FUNCTION_BLOCK FB_EventSubscriber2 IMPLEMENTS I_Observer
VAR_INPUT
	eventPublisher					: I_EventPublisher;
END_VAR
VAR
	_verbose						: BOOL := TRUE;
	_event							: INT;
	// Register after online change 
	registeredAtPublisher			: BOOL;

	breinit 						: BOOL; // reinit test marker
END_VAR

// Is there a valid publisher attached? 
IF eventPublisher=0	THEN
	RETURN;
END_IF

// Did we already register in the publisher?
IF NOT registeredAtPublisher	THEN
	registeredAtPublisher := eventPublisher.attach(THIS^);
END_IF

{attribute 'call_after_online_change_slot' := '0'}
METHOD PRIVATE fbreinit

(*	!!!!!!!!!!!!!!!!!!!!!!!!!!!!!!!!!
   	THIS METHOD is force called after every online change 
   	!= the fb_reinit system call that will be called after the instance of the concerned function block has been copied 
 	(during an online change after modifications in the function block declaration)

	This is necessary since both observer en observee 
	!!!!!!!!!!!!!!!!!!!!!!!!!!!!!!!!!	*)
registeredAtPublisher := FALSE;
breinit:=not breinit; // flip the test marker
END_METHOD

METHOD PRIVATE message : BOOL
VAR_INPUT
	dintArg						: DINT;
END_VAR
// Log message
IF _verbose  THEN
	ADSLOGDINT(
		msgCtrlMask := ADSLOG_MSGTYPE_HINT OR ADSLOG_MSGTYPE_LOG, // ADSLOG_MSGTYPE_ERROR OR ADSLOG_MSGTYPE_LOG, 
		msgFmtStr 	:= 'Subscriber 2 knows the value changed to %d',
		dintArg 	:= dintArg
		);
END_IF
END_METHOD

METHOD update : BOOL
// the publisher mentions an update, fetch the data
_event := eventPublisher.event;
message(TO_DINT(_event));
END_METHOD

END_FUNCTION_BLOCK

(* stored: Version 1.1.0.1, ProductVersion 3.1.4024.11
   POU FB_EventSubscriber2: Id {78948430-835f-4189-b81a-4f54b3428e0d}, SpecialFunc None
   Method fbreinit: Id {4f4019a2-6dab-4552-accd-abde4ac41c58}
   Method message: Id {89c2fe32-3b54-4706-b6a2-e8e1e9486d7b}
   Method update: Id {abb6583e-4f5d-489c-9536-8dff87c43972} *)
